FUNCTION_BLOCK FB_BlueColor IMPLEMENTS ITF_Color

METHOD applyColor : STRING
applyColor := 'blue';
END_METHOD

END_FUNCTION_BLOCK

(* stored: Version 1.1.0.1, ProductVersion 3.1.4024.12
   POU FB_BlueColor: Id {432a97f9-e25e-42cf-acbd-9c7a51e79fc6}, SpecialFunc None
   Method applyColor: Id {3a887440-f4bf-42e1-b147-1d5cbeade052} *)
